FUNCTION_BLOCK TcoTaskPlcExecTest EXTENDS TcoCore.TcoTask
VAR
    _isBusy : BOOL;
    _isError : BOOL;
    _isDone : BOOL;
    _isReady : BOOL;
    _isInvokeRequestTrue : BOOL;
    _counterSetValue : ULINT;
    _counterValue : ULINT;
    _invokeCounter : ULINT;
    _executeCounter : ULINT;
    _doneCounter : ULINT;
    _invokeRisingEdgeCounter : ULINT;
    _executeRisingEdgeCounter : ULINT;
    _doneRisingEdgeCounter : ULINT;
    _previousState : eTaskState;
    _counterValuePV : ULINT;
    _myIdentity : ULINT;
    _myContextIdentity : ULINT;
    _myContextStartCount : ULINT;
    _myContextEndCount : ULINT;
    _myParentIdentity : ULINT;
    _autoRestoreByMyParentEnabled : BOOL;
    _onErrorCounter : ULINT;
    _whileErrorCounter : ULINT;
    _onStartCounter : ULINT;
END_VAR

IF(THIS^._taskState = eTaskState.Requested) THEN
	_invokeCounter := _invokeCounter + 1; 
END_IF;

IF(THIS^._taskState = eTaskState.Requested AND _PreviousState <> eTaskState.Requested) THEN
	_counterValue	:=	_counterSetValue;
	_counterValuePV := _counterValue;
	_invokeRisingEdgeCounter := _invokeRisingEdgeCounter + 1;
END_IF

IF(THIS^._taskState = eTaskState.Busy AND _previousState <> eTaskState.Busy) THEN
	_executeRisingEdgeCounter := _executeRisingEdgeCounter + 1;
END_IF

_previousState	:=	THIS^._taskState;

IF(Execute()) THEN
	_executeCounter := _executeCounter + 1;	
	_counterValue := _counterValue - 1;
	DoneWhen(_counterValue <= 0);			
	ThrowWhen(ABS(_counterValuePV -_counterValue) > 1);
	_CounterValuePV := _counterValue;
END_IF

IF(THIS^._taskState = eTaskState.Done) THEN
	_doneCounter := _doneCounter + 1; 
END_IF;

IF(THIS^._taskState = eTaskState.Done AND _previousState <> eTaskState.Done) THEN
	_doneRisingEdgeCounter := _doneRisingEdgeCounter + 1; 
END_IF

{attribute 'TcRpcEnable'}
METHOD INTERNAL _GetMessage : STRING
_GetMessage := SUPER^._messenger._mime.Text;
END_METHOD

{attribute 'TcRpcEnable'}
METHOD INTERNAL _PostMessage
VAR_INPUT
	Message	:	STRING;
END_VAR
THIS^.Messenger.Post(Message ,eMessageCategory.Error);
END_METHOD

{attribute 'TcRpcEnable'}
METHOD INTERNAL _TriggerAbort
THIS^.Abort();
END_METHOD

{attribute 'TcRpcEnable'}
METHOD INTERNAL _TriggerInvoke
THIS^.Invoke();
END_METHOD

{attribute 'TcRpcEnable'}
METHOD INTERNAL _TriggerRestore
THIS^.Restore();
END_METHOD

PROPERTY CounterValue : ULINT
GET
CounterValue := _counterValue;
END_GET
SET
_counterValue := CounterValue;
END_SET
END_PROPERTY

METHOD PROTECTED OnError
_onErrorCounter := _onErrorCounter +1;
END_METHOD

METHOD PROTECTED OnStart
_onStartCounter := _onStartCounter +1;
END_METHOD

{attribute 'TcRpcEnable'}
METHOD INTERNAL ReadOutAutoRestoreProperties
_autoRestoreByMyParentEnabled	:= THIS^.AutoRestorable;
END_METHOD

{attribute 'TcRpcEnable'}
METHOD INTERNAL ReadOutIdentities
_myIdentity			:=	THIS^.Identity;
 
_myContextIdentity	:=	THIS^.Context.Identity;
		
_myContextStartCount :=	THIS^.Context.StartCycleCount;
 
_myContextEndCount	:=	THIS^.Context.EndCycleCount;
 
_myParentIdentity	:=	THIS^._Parent.Identity;
END_METHOD

{attribute 'TcRpcEnable'}
METHOD INTERNAL ReadOutState
_isBusy					:=	THIS^.Busy;	
_isError				:=	THIS^.Error;	
_isDone					:=	THIS^.Done;	
_isReady				:=	THIS^.Ready;
_isInvokeRequestTrue 	:=	THIS^._invokeRequest;
END_METHOD

{attribute 'TcRpcEnable'}
METHOD INTERNAL SetInvokeRequest
THIS^._invokeRequest := TRUE;
END_METHOD

{attribute 'TcRpcEnable'}
METHOD INTERNAL SetPreviousStateToReady
THIS^._previousState := eTaskState.Ready;
END_METHOD

(*~
	<docu>
		<summary>
			Executes until task is in ```Error``` state .
		</summary>			
	</docu>	
~*)
METHOD PROTECTED WhileError
_whileErrorCounter := _whileErrorCounter + 1;
END_METHOD

END_FUNCTION_BLOCK

(* stored: Version 1.1.0.1, ProductVersion 3.1.4024.9
   POU TcoTaskPlcExecTest: Id {d999b365-8201-09a1-30da-8c11b37c430b}, SpecialFunc None
   Method _GetMessage: Id {201e3fe2-eb96-0a73-28d4-8fa22b24ff4f}
   Method _PostMessage: Id {4778a649-9ad5-08cb-1f42-6c7f946f9a4f}
   Method _TriggerAbort: Id {9fe57617-d6d6-05f4-2449-26aa905ed514}
   Method _TriggerInvoke: Id {96032824-527e-0092-0d69-6ebb53740a1a}
   Method _TriggerRestore: Id {f93d9bec-0152-0998-2912-d8114b6d47a6}
   Property CounterValue: Id {e505bc50-fd63-0f80-0e10-605aa9e813dd}
   Get Get: Id {3c6c06da-6bfb-0d32-1a54-a5d4a3d942ae}
   Set Set: Id {033d290a-4ba2-0785-0d5b-2b41b949401c}
   Method OnError: Id {866cb534-8121-0190-0d4f-704cc10d4444}
   Method OnStart: Id {c158ae0d-0fe6-07e7-25e4-c183eee4e419}
   Method ReadOutAutoRestoreProperties: Id {d092b555-5060-0663-2d25-047918cc6c34}
   Method ReadOutIdentities: Id {f605ab32-c2ff-0150-0e7f-b7644950c7bb}
   Method ReadOutState: Id {5c4c8380-7836-0f24-3c1d-f07d6d1e102d}
   Method SetInvokeRequest: Id {17b361cd-ddd4-0fec-0d2a-9bb19609db5d}
   Method SetPreviousStateToReady: Id {2cfc1f1f-be39-04b3-3412-faec45b958d5}
   Method WhileError: Id {a587ae62-137e-0fad-372e-245f2cd9a137} *)
